// TIA Portal V19 export
TYPE "LEXCHANGETRAY_typeRollerIoSignalInterface"
// configuration: LEXCHANGETRAY_typeRollerIoSignalConfigeration
// commands: LEXCHANGETRAY_typeRollerIoSignalManualCommands
// monitoring: LEXCHANGETRAY_typeRollerIoSignalProcessValues
// stored: Access Published
   STRUCT
      configuration : "LEXCHANGETRAY_typeRollerIoSignalConfigeration";
      commands { S7_SetPoint := 'True'} : "LEXCHANGETRAY_typeRollerIoSignalManualCommands";
      monitoring { S7_SetPoint := 'True'} : "LEXCHANGETRAY_typeRollerIoSignalProcessValues";
   END_STRUCT;
END_TYPE
